{attribute addProperty BoxType "EK1122-0000-0018"}
{attribute addProperty Id "Beckhoff_EP6xxxsub_EK1100EK1100_179A0949162A_0001_EP6001_0002_0020EP6001_4599C92248060A_0002_EP6001_0002_0021EP6001_4599C92248060A_0003_EP6002_0002_0016EP6002_E497E751864108A_0004_EP6002_0002_0017EP6002_6961C256864108A_0005_EP6002_0002_0018EP6002_6961C256864108A_0006_EP6002_0002_0019EP6002_6961C256864108A_0007_EP6002_0002_0020EP6002_6961C256864108A_0008_EP6002_0002_0021EP6002_6961C256864108A_0009_EP6002_0002_0023EP6002_E45E7FFD864108A_0010_EP6002_0002_0024EP6002_E45E7FFD864108A_0011_EP6090_0000_0017EP6090_C46C03A814418A_0012_EP6224_0002_0016EP6224_341CFB1D22428A_0013_EP6224_0042_0016EP6224_997CEEB225632A_0014_EP6224_2022_0016EP6224_7C2B6CA219224A_0015_EP6224_2022_0017EP6224_7C2B6CA219224A_0016_EP6224_2022_0018EP6224_193A140119224A_0017_EP6224_3022_0016EP6224_7C2B6CA219224A_0018_EP6224_3022_0017EP6224_193A140119224A_0019_EP6228_0022_0016EP6228_2A1F57FC22428A_0020_EP6228_0022_0017EP6228_2A1F57FC22428A_0021_EP6228_0022_0018EP6228_2A1F57FC22428A_0022_EP6228_0042_0016EP6228_8FEFBC8C28836A_0023_EP6228_3032_0016EP6228_2A1F57FC22428A_0024_EP6228_3132_0016EP6228_32E67ADF25632A_0025_EP6228_3142_0016EP6228_32E67ADF25632A_0026_EP6601_0002_0018EP6601_194A340D8010"}
{attribute addProperty CRC "3142012178"}
{attribute addProperty SizeInBites "11248"}
{attribute addProperty SizeInBytes "1406"}
TYPE Beckhoff_EP6xxxEK1122_BB474D12 EXTENDS EK1122_179A0949 :
STRUCT
	{attribute addProperty Name "Beckhoff_EP6xxxsub_EK1100"}
	Beckhoff_EP6xxxsub_EK1100 : EK1100_179A0949;
	{attribute addProperty Name "A_0001_EP6001_0002_0020"}
	A_0001_EP6001_0002_0020 : EP6001_4599C922;
	{attribute addProperty Name "A_0002_EP6001_0002_0021"}
	A_0002_EP6001_0002_0021 : EP6001_4599C922;
	{attribute addProperty Name "A_0003_EP6002_0002_0016"}
	A_0003_EP6002_0002_0016 : EP6002_E497E751;
	{attribute addProperty Name "A_0004_EP6002_0002_0017"}
	A_0004_EP6002_0002_0017 : EP6002_6961C256;
	{attribute addProperty Name "A_0005_EP6002_0002_0018"}
	A_0005_EP6002_0002_0018 : EP6002_6961C256;
	{attribute addProperty Name "A_0006_EP6002_0002_0019"}
	A_0006_EP6002_0002_0019 : EP6002_6961C256;
	{attribute addProperty Name "A_0007_EP6002_0002_0020"}
	A_0007_EP6002_0002_0020 : EP6002_6961C256;
	{attribute addProperty Name "A_0008_EP6002_0002_0021"}
	A_0008_EP6002_0002_0021 : EP6002_6961C256;
	{attribute addProperty Name "A_0009_EP6002_0002_0023"}
	A_0009_EP6002_0002_0023 : EP6002_E45E7FFD;
	{attribute addProperty Name "A_0010_EP6002_0002_0024"}
	A_0010_EP6002_0002_0024 : EP6002_E45E7FFD;
	{attribute addProperty Name "A_0011_EP6090_0000_0017"}
	A_0011_EP6090_0000_0017 : EP6090_C46C03A8;
	{attribute addProperty Name "A_0012_EP6224_0002_0016"}
	A_0012_EP6224_0002_0016 : EP6224_341CFB1D;
	{attribute addProperty Name "A_0013_EP6224_0042_0016"}
	A_0013_EP6224_0042_0016 : EP6224_997CEEB2;
	{attribute addProperty Name "A_0014_EP6224_2022_0016"}
	A_0014_EP6224_2022_0016 : EP6224_7C2B6CA2;
	{attribute addProperty Name "A_0015_EP6224_2022_0017"}
	A_0015_EP6224_2022_0017 : EP6224_7C2B6CA2;
	{attribute addProperty Name "A_0016_EP6224_2022_0018"}
	A_0016_EP6224_2022_0018 : EP6224_193A1401;
	{attribute addProperty Name "A_0017_EP6224_3022_0016"}
	A_0017_EP6224_3022_0016 : EP6224_7C2B6CA2;
	{attribute addProperty Name "A_0018_EP6224_3022_0017"}
	A_0018_EP6224_3022_0017 : EP6224_193A1401;
	{attribute addProperty Name "A_0019_EP6228_0022_0016"}
	A_0019_EP6228_0022_0016 : EP6228_2A1F57FC;
	{attribute addProperty Name "A_0020_EP6228_0022_0017"}
	A_0020_EP6228_0022_0017 : EP6228_2A1F57FC;
	{attribute addProperty Name "A_0021_EP6228_0022_0018"}
	A_0021_EP6228_0022_0018 : EP6228_2A1F57FC;
	{attribute addProperty Name "A_0022_EP6228_0042_0016"}
	A_0022_EP6228_0042_0016 : EP6228_8FEFBC8C;
	{attribute addProperty Name "A_0023_EP6228_3032_0016"}
	A_0023_EP6228_3032_0016 : EP6228_2A1F57FC;
	{attribute addProperty Name "A_0024_EP6228_3132_0016"}
	A_0024_EP6228_3132_0016 : EP6228_32E67ADF;
	{attribute addProperty Name "A_0025_EP6228_3142_0016"}
	A_0025_EP6228_3142_0016 : EP6228_32E67ADF;
	{attribute addProperty Name "A_0026_EP6601_0002_0018"}
	A_0026_EP6601_0002_0018 : EP6601_194A340D;
END_STRUCT
END_TYPE

(* stored: Version 1.2.0.0, ProductVersion 3.1.4024.9
   DUT Beckhoff_EP6xxxEK1122_BB474D12: Id {1d4f5b87-08be-48e5-829c-f8bf1791e379} *)
